Fanuc KAREL source: kt00589.KL

-- PROVISIONAL review KL for V1013-1; original PC SHA256 9e4d99dc2e19ff9021e3615e90b146ebb6be4e6298896e9e9116268eb68eb390
-- Incomplete behavior may be omitted. Consult companion uncertainty JSON. Do not deploy.
PROGRAM KT00589
%NOLOCKGROUP
VAR
  S1 : STRING[80]
  S2 : STRING[80]
  OUT : STRING[80]
BEGIN
  -- UNRESOLVED_PC offsets 5-14; opcodes 3F,75
  -- UNRESOLVED_PC offsets 19-28; opcodes 3F,75
  -- UNRESOLVED_PC offsets 33-42; opcodes 3F,75
  -- UNRESOLVED_PC offsets 47-56; opcodes 3F,75
  -- UNRESOLVED_PC offsets 61-80; opcodes 73,73,7D,75
  -- UNRESOLVED_PC offsets 85-89; opcodes 7F
END KT00589
